Staubli VAL3: Deplacements.pgx

program Deplacements()
begin
  //Déplacement vers la position initiale du robot, sert uniquement lors des simulations
  movej(pRobotZeroPosition,flange,mNomSpeed)

  //Déplacement vers une position initiale de numérisation
  //movel(pInitialPosition, flange, mNomSpeed)
  //waitEndMove()

  while true
    //Décalage vers le haut
    movel(pInitialPositionRepos,flange,mNomSpeed)
    waitEndMove()

    //Execution d'un balayage de surface
    call BalayageSimple()
  endWhile
end
